// LS Electric XG5000 project: 동남144
// PLC NewPLC
// module base 0 slot 0: 입출력 모듈:XBC-DN/DP14E (DC 24V 입력 8점, 트랜지스터 출력 6점)

PROGRAM NewProgram (task: 스캔 프로그램)

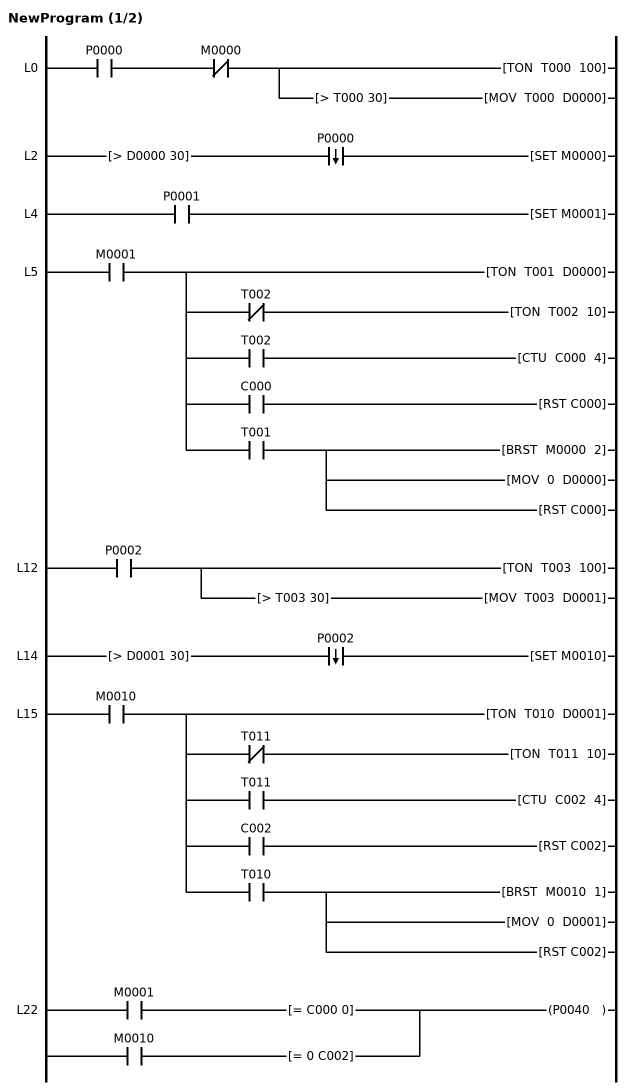
; L0
LOAD      P0000
AND NOT   M0000
TON       T000 100
AND>      T000 30
MOV       T000 D0000
; L2
LOAD>     D0000 30
ANDN      P0000
SET       M0000
; L4
LOAD      P0001
SET       M0001
; L5
LOAD      M0001
TON       T001 D0000
MPUSH
AND NOT   T002
TON       T002 10
MLOAD
AND       T002
CTU       C000 4
MLOAD
AND       C000
RST       C000
MPOP
AND       T001
BRST      M0000 2
MOV       0 D0000
RST       C000
; L12
LOAD      P0002
TON       T003 100
AND>      T003 30
MOV       T003 D0001
; L14
LOAD>     D0001 30
ANDN      P0002
SET       M0010
; L15
LOAD      M0010
TON       T010 D0001
MPUSH
AND NOT   T011
TON       T011 10
MLOAD
AND       T011
CTU       C002 4
MLOAD
AND       C002
RST       C002
MPOP
AND       T010
BRST      M0010 1
MOV       0 D0001
RST       C002
; L22
LOAD      M0001
AND=      C000 0
LOAD      M0010
AND=      0 C002
OR LOAD
OUT       P0040

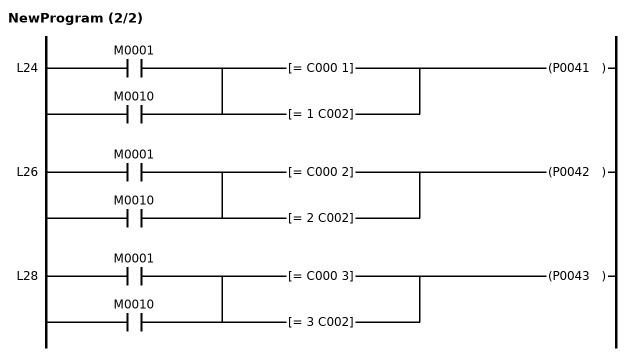
; L24
LOAD      M0001
OR        M0010
LOAD=     C000 1
OR=       1 C002
AND LOAD
OUT       P0041
; L26
LOAD      M0001
OR        M0010
LOAD=     C000 2
OR=       2 C002
AND LOAD
OUT       P0042
; L28
LOAD      M0001
OR        M0010
LOAD=     C000 3
OR=       3 C002
AND LOAD
OUT       P0043